{attribute 'qualified_only'}
VAR_GLOBAL
	Power: BOOL := FALSE;
	initialiseren:BOOL := FALSE;
	Initialisatie_voltooid: BOOL := FALSE;
	Status: STRING (INT#30):= 'OFF';
	MotorInvoer: BOOL := 0;
	ZaagLengte: INT :=0;
	HuidigePositieAanvoer: INT := 200;
	StartAanvoer: BOOL;
	AanvoerInPositie: BOOL;
	ZagenKlaar: BOOL;
	motoruitvoer: BOOL;
END_VAR

(* stored: Version 1.1.0.1, ProductVersion 3.1.4024.12
   GVL GVL: Id {54771d00-2194-439f-8002-493f6818a753} *)
